{library PUBLIC}
(* Function to get gantry status.
    This function can run continuously and will not block other communications.   
 *)
FUNCTION_BLOCK GantryStatus
VAR_INPUT
	En: 					BOOL:=FALSE;			(* Set to true to ask for status, the block  will continuously ask for status while true *)
END_VAR
VAR_OUTPUT
	Done: 					BOOL:=FALSE;			(* If true, the STATUS command is running, to stop/pause set En to false *)
	Status:					GANTRY_STATUS;			(* Gantry status *)
END_VAR
VAR_IN_OUT
	Data: 					CommunicationData;		(* Common data structure to connect this function block to a specific Communicator block *)
END_VAR
VAR
END_VAR


IF En THEN
	
	Status:=NodeReadWord(Address:=Data._Address, Channel:=2);
	Done:=TRUE;
ELSE
	Status:=GANTRY_STATUS.GANTRY_STATUS_NOT_ENABLED;
	Done:=FALSE;
END_IF;

END_FUNCTION_BLOCK

(* stored: Version 1.1.0.1, ProductVersion 3.1.4024.2
   POU GantryStatus: Id {04c4f4a5-980d-4e0e-92ff-12be407972ea}, SpecialFunc None *)
